// TIA Portal V20 export
FUNCTION_BLOCK "FB_Caroussel_Voltage_Selection"   // FB10, LAD
{ S7_Optimized_Access := 'TRUE' }
// stored: MemoryReserve 100, SetENOAutomatically false
   VAR_INPUT
      Emergency_Stop_Release : Bool;
      Selected_Voltage_220V : Bool;
      Selected_Voltage_127V : Bool;
      Carousel_Voltage_Selection : SInt;
   END_VAR
   VAR_OUTPUT
      Voltage_220V_Selected : Bool;
      Voltage_127V_Selected : Bool;
   END_VAR
   VAR
      Delay_Turn_On_220V { S7_SetPoint := 'True'} : TON_TIME;
      Delay_Turn_On_127V { S7_SetPoint := 'True'} : TON_TIME;
   END_VAR
BEGIN

REGION Network 1
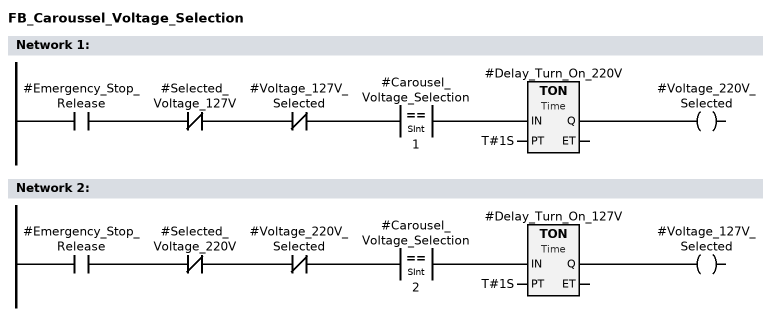
   RUNG wire#powerrail
      Contact( #Emergency_Stop_Release )
      I_Contact( #Selected_Voltage_127V )
      I_Contact( #Voltage_127V_Selected )
      { S7_Templates := "SrcType := SInt" } EQ_Contact(in1 := #Carousel_Voltage_Selection, in2 := 1)
      { S7_Templates := "time_type := Time" } #Delay_Turn_On_220V.TON(pt := T#1S, et =>)
      Coil( #Voltage_220V_Selected )
   END_RUNG
   // the same network as SCL:
   #Delay_Turn_On_220V(IN := #Emergency_Stop_Release AND NOT #Selected_Voltage_127V AND NOT #Voltage_127V_Selected AND (#Carousel_Voltage_Selection = 1),   // TON
                       PT := T#1S);
   #Voltage_220V_Selected := #Delay_Turn_On_220V.Q;
END_REGION

REGION Network 2
   RUNG wire#powerrail
      Contact( #Emergency_Stop_Release )
      I_Contact( #Selected_Voltage_220V )
      I_Contact( #Voltage_220V_Selected )
      { S7_Templates := "SrcType := SInt" } EQ_Contact(in1 := #Carousel_Voltage_Selection, in2 := 2)
      { S7_Templates := "time_type := Time" } #Delay_Turn_On_127V.TON(pt := T#1S, et =>)
      Coil( #Voltage_127V_Selected )
   END_RUNG
   // the same network as SCL:
   #Delay_Turn_On_127V(IN := #Emergency_Stop_Release AND NOT #Selected_Voltage_220V AND NOT #Voltage_220V_Selected AND (#Carousel_Voltage_Selection = 2),   // TON
                       PT := T#1S);
   #Voltage_127V_Selected := #Delay_Turn_On_127V.Q;
END_REGION
END_FUNCTION_BLOCK
